VAR_GLOBAL
{attribute 'pytmc' := 'pv: UED:SDS:SPR:A'}
{attribute 'TcLinkTo' := 	'.q_xDO1 := TIIB[Solenoid Pair A Digital IO (EP2338-0001)]^Channel 9^Output;
                          	.q_xDO2 := TIIB[Solenoid Pair A Digital IO (EP2338-0001)]^Channel 10^Output;	
'}
SolenoidPairA : FB_SolenoidPair;
	
END_VAR

(* stored: Version 1.1.0.1, ProductVersion 3.1.4024.12
   GVL GVL_MAIN: Id {e66c2fe5-8e74-49a9-9562-60ceddf31bb1} *)
